// TIA Portal V17 export
// export: Created 2023-12-22T15:05:33.1678837Z, ExportSetting WithDefaults, DisplayName Totally Integrated Automation Portal, DisplayVersion V17, DisplayName TIA Portal Openness, DisplayVersion V17, DisplayName TIA Portal Version Control Interface, DisplayVersion V17, DisplayName STEP 7 Professional, DisplayVersion V17, DisplayName STEP 7 Safety, DisplayVersion V17, DisplayName WinCC Advanced, DisplayVersion V17
DATA_BLOCK "Historian_DB"   // DB88
VERSION : 0.1
// stored: AutoNumber false, DBAccessibleFromOPCUA true, InstanceOfName Historian, InstanceOfType FB
"Historian"
   // VAR_IN_OUT
   //    Main_REQ_Start : Bool;
   //    Main_Start : Bool;
   //    HMI_Start : Bool;
   //    HMI_Stop : Bool;
   // END_VAR
   // VAR RETAIN
   //    pos : Array[0..15] of Bool;
   //    update : Bool;
   //    CMD : Bool := true;
   //    CODE : Int;
   //    DTL : DTL;
   //    LOG { S7_SetPoint := 'True'} : "Historian_LOG";
   // END_VAR
BEGIN
END_DATA_BLOCK
